// TIA Portal V17 export
// export: Created 2022-07-05T08:49:26.1285336Z, ExportSetting WithDefaults, DisplayName Totally Integrated Automation Portal, DisplayVersion V17, DisplayName TIA Portal Openness, DisplayVersion V17, DisplayName TIA Portal Version Control Interface, DisplayVersion V17, DisplayName STEP 7 Professional, DisplayVersion V17, DisplayName STEP 7 Safety, DisplayVersion V17, DisplayName WinCC Advanced, DisplayVersion V17
TYPE "typeOPCUAMethodHandling"
// stored: IsFailsafeCompliant false
   STRUCT
      Called : Bool;
      Finished : Bool;
      Result : DWord;
   END_STRUCT;
END_TYPE
